Fanuc KAREL source: ka00142.KL

-- PROVISIONAL review KL for V1013-1; original PC SHA256 8449994b0814194f3fdf8fa9c3fba80d3ca479adf936e5c0cd9319b9e587b344
-- Incomplete behavior may be omitted. Consult companion uncertainty JSON. Do not deploy.
PROGRAM KA00142
%NOLOCKGROUP
-- UNRESOLVED_DECL SRC type=002017
-- UNRESOLVED_DECL DST type=00001c
BEGIN
  -- UNRESOLVED_PC offsets 5-19; opcodes 2E,22,9D,33,B4
  -- UNRESOLVED_PC offsets 24-39; opcodes 22,9D,33,B3,23
  -- UNRESOLVED_PC offsets 44-48; opcodes 7F
END KA00142
